// TwinCAT 3 PLC project Virtual_PLC
// ProgramVersion: 3.1.4024.0
// libraries:
//   Tc2_Standard, * (Beckhoff Automation GmbH)
//   Tc2_System, * (Beckhoff Automation GmbH)
//   Tc3_Module, * (Beckhoff Automation GmbH)
// project tree:
//   GVLs/ GVL_Main.TcGVL
//   POUs/ calcTravelTime.TcPOU, PRG_BuyCoffee.TcPOU, PRG_TravelToSchool.TcPOU
//   / Task_Coffee.TcTTO, Task_Travel.TcTTO

CONFIGURATION Virtual_PLC
    RESOURCE PLC ON TwinCAT3
        TASK Task_Coffee(INTERVAL := T#10ms, PRIORITY := 21);
        TASK Task_Travel(INTERVAL := T#10ms, PRIORITY := 22);
        PROGRAM PRG_BuyCoffee WITH Task_Coffee : PRG_BuyCoffee;
        PROGRAM PRG_TravelToSchool WITH Task_Travel : PRG_TravelToSchool;
    END_RESOURCE
END_CONFIGURATION

// ---- GVLs/GVL_Main.TcGVL
{attribute 'qualified_only'}
VAR_GLOBAL
	// Communicatie tussen tasks
    coffeeReady : BOOL := FALSE;       // Wordt TRUE zodra koffie klaar is
    travelFinished : BOOL := FALSE;    // Wordt TRUE zodra je op school bent

    // Statussen
    travelState : INT := 0;            // Huidige stap in de reis
    coffeeState : INT := 0;            // Huidige stap in het koffietraject

    // Variabelen voor functie
    distanceToSchool : INT := 15;      // km
    avgSpeed : INT := 15;              // km/h
    travelTime : INT := 0;             // minuten, output van functie

END_VAR

// ---- POUs/PRG_BuyCoffee.TcPOU
PROGRAM PRG_BuyCoffee
VAR
    localTimer : TON;
END_VAR

CASE GVL_Main.coffeeState OF

    0: // Kom winkel binnen
        localTimer(IN := TRUE, PT := T#2S);
        IF localTimer.Q THEN
            GVL_Main.coffeeState := 1;
            localTimer(IN := FALSE);
        END_IF

    1: // Bestel koffie
        localTimer(IN := TRUE, PT := T#2S);
        IF localTimer.Q THEN
            GVL_Main.coffeeState := 2;
            localTimer(IN := FALSE);
        END_IF

    2: // Wacht tot koffie klaar
        localTimer(IN := TRUE, PT := T#4S);
        IF localTimer.Q THEN
            GVL_Main.coffeeState := 3;
            localTimer(IN := FALSE);
        END_IF

    3: // Neem koffie aan
        GVL_Main.coffeeReady := TRUE;
        localTimer(IN := TRUE, PT := T#1S);
        IF localTimer.Q THEN
            GVL_Main.coffeeState := 4;
            localTimer(IN := FALSE);
        END_IF

    4: // Loop winkel uit
        // Klaar
        localTimer(IN := FALSE);
		GVL_Main.coffeeReady := TRUE;
		
END_CASE

END_PROGRAM

// ---- POUs/PRG_TravelToSchool.TcPOU
PROGRAM PRG_TravelToSchool
VAR
    localTimer : TON; // timer voor simulatie
	travelFinished: BOOL;
	travelTime: INT;
	distanceToSchool: INT;
	avgSpeed: INT;
	coffeeReady: BOOL;
END_VAR
VAR_INPUT
	travelState: INT;
END_VAR

CASE GVL_Main.travelState OF

    0: // Start
        localTimer(IN := TRUE, PT := T#2S);
        IF localTimer.Q THEN
            GVL_Main.travelState := 1;
            localTimer(IN := FALSE);
        END_IF

    1: // Stap op fiets naar station Almelo
        localTimer(IN := TRUE, PT := T#3S);
        IF localTimer.Q THEN
            GVL_Main.travelState := 2;
            localTimer(IN := FALSE);
        END_IF

    2: // Op station Almelo, instappen trein
        localTimer(IN := TRUE, PT := T#2S);
        IF localTimer.Q THEN
            GVL_Main.travelState := 3;
            localTimer(IN := FALSE);
        END_IF

    3: // In trein naar Enschede
        localTimer(IN := TRUE, PT := T#4S);
        IF localTimer.Q THEN
            GVL_Main.travelState := 4;
            localTimer(IN := FALSE);
        END_IF

    4: // Op station Enschede, begin lopen
        localTimer(IN := TRUE, PT := T#3S);
        IF localTimer.Q THEN
            GVL_Main.travelState := 5;
            localTimer(IN := FALSE);
        END_IF

    5: // Onderweg: check of koffie klaar is
        IF GVL_Main.coffeeReady THEN
            GVL_Main.travelState := 6;
        END_IF

    6: // Op school met koffie
        GVL_Main.travelFinished := TRUE;
        GVL_Main.travelTime := calcTravelTime(distanceToSchool, avgSpeed); // functie-aanroep

END_CASE

END_PROGRAM

// ---- POUs/calcTravelTime.TcPOU
FUNCTION calcTravelTime : INT
VAR_INPUT
    distance : INT; // in kilometers
    speed : INT;    // in km/h
END_VAR

// Simpele berekening reistijd in minuten
calcTravelTime := (distance) / speed;

END_FUNCTION
